PROGRAM CraneSimulation
VAR
	fInitialVelocity : REAL := 0;
	fInitialPosition : REAL := 0;
END_VAR

IF Inputs.bStartSimulation AND Inputs.bAutoMode THEN
	Outputs.fSimulationTime := Outputs.fSimulationTime + Parameters.fCyclicTime;
ELSE
	Outputs.fSimulationTime := 0;
END_IF

IF Outputs.fSimulationTime > 0 AND Inputs.bAutoMode THEN
	Parameters.bSimulationRunning := TRUE;
ELSE
	Parameters.bSimulationRunning := FALSE;
END_IF

IF Inputs.bAutoMode THEN
	Outputs.fCylinderVelocity := Inputs.fCylinderVelocityReference;
	Outputs.fCylinderPosition := Outputs.fCylinderVelocity * (Outputs.fSimulationTime*Outputs.fSimulationTime)/2 + fInitialVelocity*Outputs.fSimulationTime + fInitialPosition;
ELSE
	Outputs.fCylinderPosition := Inputs.fManualCylinderPositionReference;
END_IF

END_PROGRAM

(* stored: Version 1.1.0.1, ProductVersion 3.1.4024.10
   POU CraneSimulation: Id {9db64730-0769-4523-9dc9-b42b5865fac6}, SpecialFunc None *)
